// TIA Portal project "Project13" (V15.1)

(* hardware
DEVICE "S7-1200 station_1"  S7-1200 Station
   slot 0: "Rack_0"  S7-1200 Rack  Rack  V1.0
   slot 1: "PLC_1"  CPU 1214C DC/DC/Rly  6ES7 214-1HG40-0XB0  V4.2
   slot 2: "DQ 16x24VDC_1"  6ES7 222-1BH30-0XB0  V1.0
*)

// ===== PLC "PLC_1"  CPU 1214C DC/DC/Rly =====

VAR_GLOBAL   // PLC tag table "Default tag table"
   "Start" AT %I0.0 : Bool;
   "Stop" AT %I0.1 : Bool;
   "Reset" AT %I0.2 : Bool;
   "Palet sensörü" AT %I0.3 : Bool;
   "Alt sensör" AT %I0.4 : Bool;
   "Üst Sensör" AT %I0.5 : Bool;
   "Yüklendi sensörü" AT %I0.6 : Bool;
   "Sol giriş Sensörü" AT %I0.7 : Bool;
   "Sol çıkış sensörü" AT %I1.0 : Bool;
   "Sağ giriş sensörü" AT %I1.1 : Bool;
   "Sağ çıkış sensörü" AT %I1.2 : Bool;
   "Ana konveyör" AT %Q1.3 : Bool;
   "Transfer Konveyör" AT %Q1.4 : Bool;
   "Sola Transfer" AT %Q1.5 : Bool;
   "Sağa Transfer" AT %Q1.6 : Bool;
   "Counter Ekranı" AT %QW8 : Word;
   "Sistem mem" AT %M10.0 : Bool;
   "Alt sensör Mem" AT %M10.1 : Bool;
   "sol koveyör" AT %Q10.2 : Bool;
   "sağ konveyör" AT %Q10.3 : Bool;
   "üst sensör mem" AT %M10.4 : Bool;
END_VAR

// folder: System blocks/Program resources

DATA_BLOCK "Timer1"   // DB1
{ S7_Optimized_Access := 'TRUE' }
AUTHOR : Simatic
FAMILY : IEC
NAME : IEC_TMR
VERSION : 1.0
// stored: InstanceOfName IEC_TIMER
"IEC_TIMER"
BEGIN
END_DATA_BLOCK

DATA_BLOCK "Timer2"   // DB2
{ S7_Optimized_Access := 'TRUE' }
AUTHOR : Simatic
FAMILY : IEC
NAME : IEC_TMR
VERSION : 1.0
// stored: InstanceOfName IEC_TIMER
"IEC_TIMER"
BEGIN
END_DATA_BLOCK

// folder: (top level)

ORGANIZATION_BLOCK "Main"   // OB1, LAD, ProgramCycle
TITLE = "Main Program Sweep (Cycle)"
{ S7_Optimized_Access := 'TRUE' }
VERSION : 0.1
   VAR_INPUT
      Initial_Call : Bool;   // Initial call of this OB
      Remanence : Bool;   // =True, if remanent data are available
   END_VAR
BEGIN

REGION Network 1
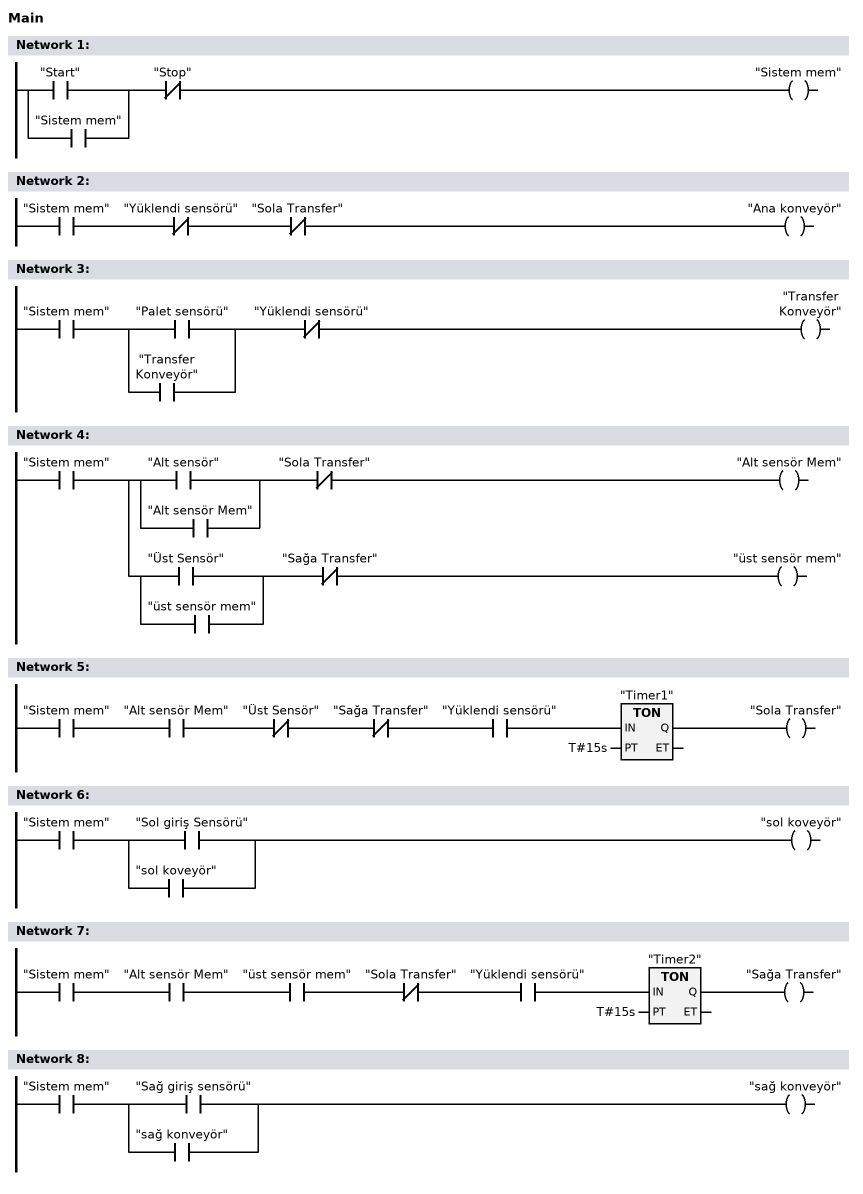
   RUNG wire#powerrail
      Contact( "Start" )
      wire#w1
      I_Contact( "Stop" )
      Coil( "Sistem mem" )
   END_RUNG
   RUNG wire#powerrail
      Contact( "Sistem mem" )
   END_RUNG wire#w1
   // the same network as SCL:
   "Sistem mem" := ("Start" OR "Sistem mem") AND NOT "Stop";
END_REGION

REGION Network 2
   RUNG wire#powerrail
      Contact( "Sistem mem" )
      I_Contact( "Yüklendi sensörü" )
      I_Contact( "Sola Transfer" )
      Coil( "Ana konveyör" )
   END_RUNG
   // the same network as SCL:
   "Ana konveyör" := "Sistem mem" AND NOT "Yüklendi sensörü" AND NOT "Sola Transfer";
END_REGION

REGION Network 3
   RUNG wire#powerrail
      Contact( "Sistem mem" )
      wire#w1
      Contact( "Palet sensörü" )
      wire#w2
      I_Contact( "Yüklendi sensörü" )
      Coil( "Transfer Konveyör" )
   END_RUNG
   RUNG wire#w1
      Contact( "Transfer Konveyör" )
   END_RUNG wire#w2
   // the same network as SCL:
   "Transfer Konveyör" := "Sistem mem" AND ("Palet sensörü" OR "Transfer Konveyör") AND NOT "Yüklendi sensörü";
END_REGION

REGION Network 4
   RUNG wire#powerrail
      Contact( "Sistem mem" )
      wire#w1
      Contact( "Alt sensör" )
      wire#w2
      I_Contact( "Sola Transfer" )
      Coil( "Alt sensör Mem" )
   END_RUNG
   RUNG wire#w1
      Contact( "Alt sensör Mem" )
   END_RUNG wire#w2
   RUNG wire#w1
      Contact( "Üst Sensör" )
      wire#w3
      I_Contact( "Sağa Transfer" )
      Coil( "üst sensör mem" )
   END_RUNG
   RUNG wire#w1
      Contact( "üst sensör mem" )
   END_RUNG wire#w3
   // the same network as SCL:
   "Alt sensör Mem" := "Sistem mem" AND ("Alt sensör" OR "Alt sensör Mem") AND NOT "Sola Transfer";
   "üst sensör mem" := "Sistem mem" AND ("Üst Sensör" OR "üst sensör mem") AND NOT "Sağa Transfer";
END_REGION

REGION Network 5
   "Timer1".TON(IN := "Sistem mem" AND "Alt sensör Mem" AND NOT "Üst Sensör" AND NOT "Sağa Transfer" AND "Yüklendi sensörü",
                PT := T#15s);
   "Sola Transfer" := "Timer1".Q;
END_REGION

REGION Network 6
   RUNG wire#powerrail
      Contact( "Sistem mem" )
      wire#w1
      Contact( "Sol giriş Sensörü" )
      wire#w2
      Coil( "sol koveyör" )
   END_RUNG
   RUNG wire#w1
      Contact( "sol koveyör" )
   END_RUNG wire#w2
   RUNG wire#powerrail
   END_RUNG
   // the same network as SCL:
   "sol koveyör" := "Sistem mem" AND ("Sol giriş Sensörü" OR "sol koveyör");
END_REGION

REGION Network 7
   "Timer2".TON(IN := "Sistem mem" AND "Alt sensör Mem" AND "üst sensör mem" AND NOT "Sola Transfer" AND "Yüklendi sensörü",
                PT := T#15s);
   "Sağa Transfer" := "Timer2".Q;
END_REGION

REGION Network 8
   RUNG wire#powerrail
      Contact( "Sistem mem" )
      wire#w1
      Contact( "Sağ giriş sensörü" )
      wire#w2
      Coil( "sağ konveyör" )
   END_RUNG
   RUNG wire#w1
      Contact( "sağ konveyör" )
   END_RUNG wire#w2
   // the same network as SCL:
   "sağ konveyör" := "Sistem mem" AND ("Sağ giriş sensörü" OR "sağ konveyör");
END_REGION
END_ORGANIZATION_BLOCK